{attribute 'linkalways'} 
{attribute 'no_explicit_call' := 'This FB is a CLASS and must be accessed using methods or properties'}
{attribute 'enable_dynamic_creation'}
FUNCTION_BLOCK _ETcVnNbc EXTENDS EnumDatatypeBase
VAR
	localData : ETcVnNbc;
	activeData : REFERENCE TO ETcVnNbc;
	enumBaseDatatype : _UDINT(localData);
END_VAR

METHOD PRIVATE AddLocalEnumeration
VAR_INPUT
	Enumeration : T_MAXSTRING;
	Value : ETcVnNbc;
END_VAR
AddEnumeration(Enumeration, Value);
END_METHOD

PROPERTY PUBLIC Address : PVOID
GET
Address := ADR(activeData);
END_GET
END_PROPERTY

METHOD PUBLIC ClearReference
VAR_INPUT
END_VAR
activeData REF= localData;
SetBaseDatatypeReference();
END_METHOD

METHOD PUBLIC Clone : I_Datatype
VAR
    pClone : POINTER TO _ETcVnNbc;
END_VAR
pClone := __NEW(_ETcVnNbc(InitialValue := Value));
Clone := pClone^;
END_METHOD

METHOD FB_init : BOOL
VAR_INPUT
	bInitRetains : BOOL; // if TRUE, the retain variables are initialized (warm start / cold start)
	bInCopyCode : BOOL;  // if TRUE, the instance afterwards gets moved into the copy code (online change)
	InitialValue : ETcVnNbc;
END_VAR
localData := InitialValue;
AddBaseDatatype(enumBaseDatatype);
ClearReference();

AddLocalEnumeration('TCVN_NBC_CLASSIFIER', ETcVnNbc.TCVN_NBC_CLASSIFIER);
AddLocalEnumeration('TCVN_NBC_NOVELTY_DETECTOR', ETcVnNbc.TCVN_NBC_NOVELTY_DETECTOR);
END_METHOD

PROPERTY PUBLIC Identifier : T_MAXSTRING
GET
Identifier := 'ETcVnNbc';
END_GET
END_PROPERTY

METHOD IsEnumeratorValueEqual : BOOL
VAR_INPUT
	Enumerator : I_KeyValueForwardEnumerator;
END_VAR
VAR
	storedValue : ETcVnNbc;
END_VAR
IF NOT Enumerator.TryGet(storedValue) THEN
	RETURN;
END_IF

IsEnumeratorValueEqual := storedValue = activeData;
END_METHOD

METHOD PUBLIC MakeReferenceTo
VAR_INPUT
	ReferenceTarget : REFERENCE TO ETcVnNbc;
END_VAR
activeData REF= ReferenceTarget;
SetBaseDatatypeReference();
END_METHOD

METHOD PROTECTED SetBaseDatatypeReference
VAR_INPUT
END_VAR
enumBaseDatatype.MakeReferenceTo(activeData);
END_METHOD

PROPERTY PUBLIC Size : UDINT
GET
Size := SIZEOF(activeData);
END_GET
END_PROPERTY

METHOD TryMakeReferenceTo : BOOL
VAR_INPUT
	Target : I_Datatype;
END_VAR
VAR
	targetAsEnum : I_EnumDatatype;
	pTargetData : POINTER TO ETcVnNbc;
END_VAR
IF NOT Target.TryResolveAsEnumDatatype(targetAsEnum) THEN
	RETURN;
END_IF

IF targetAsEnum.Identifier <> Identifier THEN
	RETURN;
END_IF

pTargetData := Target.Address;
activeData REF= pTargetData^;
SetBaseDatatypeReference();
TryMakeReferenceTo := TRUE;
END_METHOD

PROPERTY PUBLIC Value : ETcVnNbc
GET
Value := activeData;
END_GET
SET
activeData := Value;
END_SET
END_PROPERTY

END_FUNCTION_BLOCK

(* stored: Version 1.1.0.1, ProductVersion 3.1.4024.12
   POU _ETcVnNbc: Id {a645f0f2-fea4-4730-802c-341af3e55c08}, SpecialFunc None
   Folder Constructor: Id {0b2d8b37-8785-4c55-955e-f58c82d87dc8}
   Folder Private: Id {308f1a55-242e-4f7b-8b2d-0bb2c0416a84}
   Folder Protected: Id {d5d88e69-5978-4847-a781-13e0e796caef}
   Method AddLocalEnumeration: Id {fd8a16cf-73f1-47e0-9d43-c295e4d8c68a}
   Property Address: Id {b1dc7574-2649-4a4d-b1a2-191e5c4478f4}
   Get Get: Id {f8f27486-2d2d-41d5-8f78-8d1e176245f0}
   Method ClearReference: Id {0006c7ca-a76e-4095-abb0-6490f256e8fe}
   Method Clone: Id {e18cdebc-36c8-48fb-a548-c06bf2baa0fc}
   Method FB_init: Id {e2138ade-35ac-441f-b8c5-25cf39268389}
   Property Identifier: Id {ad9b411d-f607-4951-a994-898d94494fef}
   Get Get: Id {db90e1e4-9c6d-4848-ac10-a2634aafff58}
   Method IsEnumeratorValueEqual: Id {93c58dda-e258-46ee-8f8e-65152b6cbe65}
   Method MakeReferenceTo: Id {00540b2d-db73-49f5-bfda-3c5bd94885d5}
   Method SetBaseDatatypeReference: Id {30cf56d7-b34c-4dc6-9fda-a08fe174fa60}
   Property Size: Id {88200054-a9ea-4848-8137-0516f6407b9f}
   Get Get: Id {dae23b8e-0e37-46a3-938a-d73b80d66578}
   Method TryMakeReferenceTo: Id {fef5faa4-bf96-4ab4-b016-bc20a4e9c693}
   Property Value: Id {11891a02-2293-44e3-8968-aaf8a6652904}
   Get Get: Id {b8f61622-a7b6-4c99-8a3b-da5d69ad3dce}
   Set Set: Id {9a736a0c-fce5-48c5-a2af-ec7fe8cdb11a} *)
